TYPE stDevBase :
STRUCT
	sTagName : STRING;
	sDescription : STRING;
END_STRUCT
END_TYPE

(* stored: Version 1.1.0.1, ProductVersion 3.1.4024.12
   DUT stDevBase: Id {a5a3699e-90d5-4ff4-b090-c94bdc753e53} *)
